PROGRAM MAIN
VAR
END_VAR

END_PROGRAM

(* stored: Version 1.1.0.1
   POU MAIN: Id {34727174-fd0e-47d3-bee5-dbb1f2c016f8} *)
